# B&R Automation Studio project Semafor
Automation Studio 4.9.2.46; technology packages: Acp10Arnc0 5.12.2

## Configuration Config1

CPU X20CP3585, AutomationRuntime C4.90, Build 4.1.2, Vc V4.72.2

### Task classes (Cpu.sw)
```
Cyclic#4:
  Semafor <- Semafor.prg
VcDataObjects: Visu <- Visu.dob
Binaries: udbdef, FWRules, TCData, iomap, ashwac, Role, sysconf, arconfig, asfw, User, ashwd
Libraries: SemaforLib
```

### Hardware
```
X20CP3585 : X20CP3585 v1.8.1.0
  Connector IF2:
    ActivateDevice = 1
    Mode = Manual
    InternetAddress = 127.0.0.1
    Vnc1
    VncVcObjectName1 = Visu
    VncKeyMappingFile1 = VC\PS2-Keyboard.dis
  ConfigurationID = Semafor_Config1
  Simulation = 1
```

- Physical/Config1/X20CP3585/IoMap.iom: same as Physical/Config1/X20CP3585/Cpu.per
- Physical/Config1/X20CP3585/PvMap.vvm: same as Physical/Config1/X20CP3585/Cpu.per
- Safety project (password-protected, skipped)

## Logical view

Binary libraries used (declarations not repeated): runtime, operator, astime, AsIecCon, sys_lib, standard, io_lib, SafeMC 5.12.2, Acp10man 5.12.2, Acp10par 5.12.2, NcGlobal 5.12.2, LoopConR 4.10.2, brsystem

### Global.var - Global variables
```iecst
VAR

	WalkRequest : {REDUND_UNREPLICABLE} BOOL := FALSE; (* tlacítko pro požadavek na prejití silnice *)
	AutoWalkPeriod : {REDUND_UNREPLICABLE} TIME := T#60s; (* perioda pro automatické zapnutí prechodu *)
	WalkingTime : {REDUND_UNREPLICABLE} TIME := T#10s; (* cas aktivní zelené pro prechod chodce  *)
	Red4Car : {REDUND_UNREPLICABLE} BOOL; (* cervená na semaforu pro auta *)
	Amber4Car : {REDUND_UNREPLICABLE} BOOL; (* žlutá na semaforu pro auta *)
	Green4Car : {REDUND_UNREPLICABLE} BOOL; (* zelená na semaforu pro auta *)
	Red4Walk : {REDUND_UNREPLICABLE} BOOL; (* cervená na semaforu pro chodce *)
	Green4Walk : {REDUND_UNREPLICABLE} BOOL; (* zelená na semaforu pro chodce *)
END_VAR

VAR CONSTANT

END_VAR
```

### Package Logical/Libraries - Global libraries

### Library Logical/Libraries/SemaforLib (IEC)

#### Types.typ - Exported data types
```iecst
TYPE
	CarLightType : 	STRUCT
		State : INT := 0; (* State : 0 = init, 1 = carWay, 2 = walkWay  *)
		CarWayEna : BOOL := TRUE;
		WalkWayEna : BOOL := FALSE;
	END_STRUCT;

	WalkLightType : STRUCT
		state : INT := 0; (* State : 0 = init, 1 = WalkClosed, 2 = WalkOpen*)
		WalkEna : BOOL := FALSE; (* *)
	END_STRUCT;

	ColorStatusType : STRUCT
		RED : INT:= 0;
		AMBER : INT:= 0;
		GREEN : INT:= 0;
	END_STRUCT;

END_TYPE
```

#### SemaforLib.fun - Exported functions and function blocks
```iecst
{REDUND_ERROR} FUNCTION_BLOCK CarLight (*TODO: Add your comment here*) (*$GROUP=User,$CAT=User,$GROUPICON=User.png,$CATICON=User.png*)
	VAR_INPUT
		WalkRequest : {REDUND_UNREPLICABLE} BOOL := FALSE; (* tlacítko pro požadavek na prejití silnice *)
		AutoWalkPeriod : {REDUND_UNREPLICABLE} TIME := T#60s; (* perioda pro automatické zapnutí prechodu *)
		CarLightEna : {REDUND_UNREPLICABLE} BOOL := FALSE; (* Start state machine *)
	END_VAR
	VAR_OUTPUT
		Red4Car : {REDUND_UNREPLICABLE} BOOL; (* cervená na semaforu pro auta *)
		Amber4Car : {REDUND_UNREPLICABLE} BOOL; (* žlutá na semaforu pro auta *)
		Green4Car : {REDUND_UNREPLICABLE} BOOL; (* zelená na semaforu pro auta *)
		CarWayClosed : {REDUND_UNREPLICABLE} BOOL; (* Signal uzavrení cesty pro auta *)
	END_VAR
	VAR
		StateChangeEnable : {REDUND_UNREPLICABLE} BOOL;
		StateChangeTime : {REDUND_UNREPLICABLE} TIME := T#5s;
		TonWalkingTime : {REDUND_UNREPLICABLE} TON;
		TonStateChange : {REDUND_UNREPLICABLE} TON;
		SemaforCtrl : {REDUND_UNREPLICABLE} CarLightType;
		TofFlashing : TOF;
		TonFlashing : TON;
		ColorStatus : ColorStatusType;
		MinRequestTime : {REDUND_UNREPLICABLE} TIME := T#10s;
	END_VAR
END_FUNCTION_BLOCK

{REDUND_ERROR} FUNCTION_BLOCK WalkLight (*TODO: Add your comment here*) (*$GROUP=User,$CAT=User,$GROUPICON=User.png,$CATICON=User.png*)
	VAR_INPUT
		LightEna : {REDUND_UNREPLICABLE} BOOL; (*Start state machine*)
		WalkingTime : {REDUND_UNREPLICABLE} TIME := T#10s; (* cas aktivní zelené pro prechod chodce  *)
	END_VAR
	VAR_OUTPUT
		Red4Walk : {REDUND_UNREPLICABLE} BOOL; (* cervená na semaforu pro chodce *)
		Green4Walk : {REDUND_UNREPLICABLE} BOOL; (* zelená na semaforu pro chodce *)
		WalkClosed : {REDUND_UNREPLICABLE} BOOL; (* konec state machine *)
	END_VAR
	VAR
		WalkLightCtrl : {REDUND_UNREPLICABLE} WalkLightType;
		ColorStatus : ColorStatusType;
		TonWalkingTime : {REDUND_UNREPLICABLE} TON;
	END_VAR
END_FUNCTION_BLOCK
```

#### CarLight.st
```iecst
(* TODO: Add your comment here *)
FUNCTION_BLOCK CarLight

		// State machine
		Red4Car := FALSE;
		Amber4Car := FALSE;
		Green4Car := FALSE;
		CarWayClosed := FALSE;

	// Way closing
	IF (SemaforCtrl.State = 4) THEN
		Amber4Car := TRUE;
		StateChangeEnable := TRUE;
		ColorStatus.RED := 7;
		ColorStatus.AMBER := 42;
		ColorStatus.GREEN := 7;
		//Transition
		IF TonStateChange.Q THEN
			SemaforCtrl.State := 1;
			ColorStatus.AMBER := 7;
		END_IF;
	END_IF;

	// Way Open
	IF (SemaforCtrl.State = 3) THEN
		Green4Car := TRUE;
		StateChangeEnable := TRUE;
		ColorStatus.RED := 7;
		ColorStatus.AMBER := 7;
		ColorStatus.GREEN := 215;
		//Transition
		IF TonStateChange.Q OR (TonStateChange.ET > (AutoWalkPeriod - MinRequestTime ) AND WalkRequest) THEN
			SemaforCtrl.State := 4;
			StateChangeTime:= T#5s;
		END_IF;
	END_IF;

	// Way opening
	IF (SemaforCtrl.State = 2) THEN
		Red4Car := TRUE;
		Amber4Car := TRUE;
		StateChangeEnable := TRUE;
		ColorStatus.RED := 51;
		ColorStatus.AMBER := 42;
		ColorStatus.GREEN := 7;
		//Transition
		IF TonStateChange.Q THEN
			ColorStatus.AMBER := 7;
			SemaforCtrl.State := 3;
			StateChangeTime:= AutoWalkPeriod;
		END_IF;
	END_IF;

	// Way Closed
	IF (SemaforCtrl.State = 1) THEN
		Red4Car := TRUE;
		CarWayClosed := TRUE;
		ColorStatus.RED := 51;
		ColorStatus.AMBER := 7;
		ColorStatus.GREEN := 7;
		//Transition
		IF CarLightEna THEN
			ColorStatus.RED := 7;
			SemaforCtrl.State := 2;
			StateChangeTime:= T#3s;

		END_IF;
	END_IF;

	// Init state Amber flashing
	IF SemaforCtrl.State = 0 THEN
		//startTimerEna
		Amber4Car := TonFlashing.Q;
		StateChangeEnable := TRUE;
		StateChangeTime := T#10s;
		ColorStatus.RED := 7;
		ColorStatus.AMBER := 7;
		ColorStatus.GREEN := 7;
		//Transition
		IF TonStateChange.Q THEN
			SemaforCtrl.State := 1;
		END_IF;
	END_IF;
	// Transition Timer reset
	IF TonStateChange.Q THEN
		StateChangeEnable := FALSE;
	END_IF;

	TonStateChange(IN:=StateChangeEnable, PT:= StateChangeTime);

	TonFlashing(IN:= NOT TofFlashing.Q, PT:=T#500ms);
	TofFlashing(IN:= NOT TonFlashing.Q, PT:=T#500ms);

END_FUNCTION_BLOCK
```

#### WalkLight.st
```iecst
(* TODO: Add your comment here *)
FUNCTION_BLOCK WalkLight

	Red4Walk := FALSE;
	Green4Walk := FALSE;
	WalkLightCtrl.WalkEna := FALSE;
	WalkClosed := FALSE;

	// init lights off
	IF WalkLightCtrl.state = 0 THEN
		ColorStatus.RED := 0;
		ColorStatus.GREEN := 0;
		IF LightEna THEN
			WalkLightCtrl.state := 1;
		END_IF;
	END_IF;

	// Walk closed
	IF WalkLightCtrl.state = 1 THEN
		Red4Walk := TRUE;
		ColorStatus.RED := 51;
		ColorStatus.GREEN := 7;
		IF LightEna THEN
			WalkLightCtrl.state := 2;
		END_IF;
	END_IF;

	// Walk open
	IF WalkLightCtrl.state = 2 THEN
		Green4Walk := TRUE;
		WalkLightCtrl.WalkEna := TRUE;
		ColorStatus.RED := 7;
		ColorStatus.GREEN := 215;
		IF TonWalkingTime.Q THEN
			WalkLightCtrl.state := 1;
			WalkClosed := TRUE;
		END_IF;
	END_IF;

	//Timer
	TonWalkingTime(IN:=WalkLightCtrl.WalkEna, PT:= WalkingTime);
	WalkClosed := TonWalkingTime.Q;

END_FUNCTION_BLOCK
```

### Program Logical/Semafor (IEC)

#### Main.st - Init, cyclic, exit code
```iecst
PROGRAM _INIT
	(* Insert code here *)

END_PROGRAM

PROGRAM _CYCLIC

	// Walk light
	WalkLight_Inst0(LightEna := CarLight_Inst0.CarWayClosed, WalkingTime := WalkingTime);
	Red4Walk := WalkLight_Inst0.Red4Walk;
	Green4Walk := WalkLight_Inst0.Green4Walk;

	// Car Light
	CarLight_Inst0(CarLightEna:= WalkLight_Inst0.WalkClosed,WalkRequest:= WalkRequest,AutoWalkPeriod := AutoWalkPeriod);
	Red4Car := CarLight_Inst0.Red4Car;
	Amber4Car := CarLight_Inst0.Amber4Car;
	Green4Car := CarLight_Inst0.Green4Car;
END_PROGRAM

PROGRAM _EXIT
	(* Insert code here *)

END_PROGRAM
```

#### Variables.var - Local variables
```iecst
(**********************)

VAR
	WalkLight_Inst0 : WalkLight;
	CarLight_Inst0 : CarLight;
END_VAR
```

- Visualisation Logical/Visu (not shown)
